# EPICS autosave request: pointGreyApp/Db/pointGreyProperty_settings.req
$(P)$(R)$(PROPERTY)Val
$(P)$(R)$(PROPERTY)AutoMode
